PROGRAM MAIN
VAR
END_VAR

END_PROGRAM

(* stored: Version 1.1.0.1
   POU MAIN: Id {0adcd89b-82e2-431e-8ae9-edc53878323a} *)
